{attribute 'Tc2GvlVarNames'}
VAR_CONFIG
END_VAR

(* stored: Version 1.1.0.1, ProductVersion 3.1.4022.12
   GVL Variable_Configuration: Id {6d65dc97-d2dc-4d80-9a1f-d52333eed82a} *)
